# EPICS autosave request: supportCode/op/autosave/SPCe_settings.req
%
% Gamma SPCe ion pump power supplies
%
% vacuum pressure alarms
$(P).LOLO
$(P).LOW
$(P).HIGH
$(P).HIHI
